(* Logix 5000 project; controller Ex_2_15 Emulate 5570 rev 33.11; software revision 33.00 *)
// Program for a cooker hood

TASK MainTask (continuous, watchdog 500 ms) : MainProgram

MODULES
   Local : Emulate 5570 (ICP 4, rev 33.11)
END_MODULES

VAR_GLOBAL   (* controller tags *)
   Fan_High_Speed : BOOL;
   Fan_Low_Speed : BOOL;
   Fan_Mid_Speed : BOOL;
   Fan_Off : BOOL;
   Fan_On : BOOL;
   Light_off : BOOL;
   Light_on : BOOL;
   Ons_1 : BOOL;
   ons_2 : BOOL;
   ONS_3 : BOOL;
   S1 : BOOL;   // Fan at Low speed
   S2 : BOOL;   // Fan at Medium speed
   S3 : BOOL;   // Fan at High speed
   Switch_Fan_off : BOOL;
   Switch_Fan_on : BOOL;
   Switch_Light_Off : BOOL;   // Light off Switch
   Switch_Light_On : BOOL;   // Light On switch
END_VAR

PROGRAM MainProgram   (* main routine MainRoutine *)

ROUTINE MainRoutine   (* ladder *)
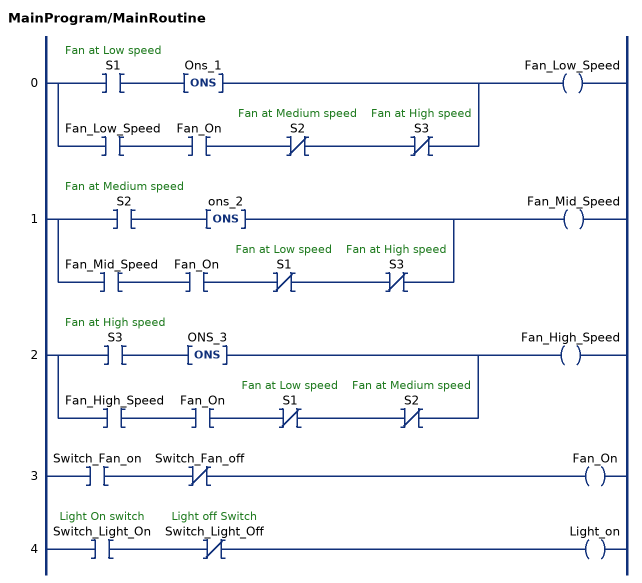
   0: [XIC(S1) ONS(Ons_1) ,XIC(Fan_Low_Speed) XIC(Fan_On) XIO(S2) XIO(S3) ]OTE(Fan_Low_Speed);
   1: [XIC(S2) ONS(ons_2) ,XIC(Fan_Mid_Speed) XIC(Fan_On) XIO(S1) XIO(S3) ]OTE(Fan_Mid_Speed);
   2: [XIC(S3) ONS(ONS_3) ,XIC(Fan_High_Speed) XIC(Fan_On) XIO(S1) XIO(S2) ]OTE(Fan_High_Speed);
   3: XIC(Switch_Fan_on)XIO(Switch_Fan_off)OTE(Fan_On);
   4: XIC(Switch_Light_On)XIO(Switch_Light_Off)OTE(Light_on);
END_ROUTINE
END_PROGRAM
